FUNCTION_BLOCK FB_Room
VAR_INPUT
	AC_IPAddr: STRING;
	ACcontrol: ST_ACcontrol;
END_VAR
VAR_OUTPUT
	ACstatus: ST_ACStatus;
END_VAR
VAR
	fbLamp : ARRAY[0..3] OF FB_Lamp;
	fbDimmer : ARRAY[0..3] OF FB_Dimmer;
	fbCurtain: FB_Curtain;
	fbAC: FB_AC;
	i: INT;
	fbAC_oop: FB_AC_oop;
END_VAR

	
	FOR i := 0 TO 3 BY 1 DO
		fbLamp[i]();
		fbDimmer[i]();
	END_FOR
	
	//fbAC(AC_IPAddr	:=	AC_IPAddr, ACcontrol:= ACcontrol, ACstatus=> ACstatus);
	fbCurtain();

END_FUNCTION_BLOCK

(* stored: Version 1.1.0.1, ProductVersion 3.1.4024.12
   POU FB_Room: Id {442c75c1-7593-4393-b6bc-5705fce27c62}, SpecialFunc None *)
